// TIA Portal V17 export
// export: Created 2024-09-02T12:50:17.7770543Z, ExportSetting WithDefaults, DisplayName Totally Integrated Automation Portal, DisplayVersion V17, DisplayName TIA Portal Openness, DisplayVersion V17, DisplayName TIA Portal Version Control Interface, DisplayVersion V17, DisplayName STEP 7 Professional, DisplayVersion V17, DisplayName STEP 7 Safety, DisplayVersion V17, DisplayName WinCC Professional, DisplayVersion V17
DATA_BLOCK "SysDI_HMI_SystemInit_OP70"   // DB259
{ DB_Accessible_From_OPC_UA := 'FALSE' }
AUTHOR : OlegFuehrus
FAMILY : HMI
NAME : HMI
VERSION : 0.1
// stored: AutoNumber true, DBAccessibleFromOPCUA false, InstanceOfName SysFB_HMI_SystemInit, InstanceOfType FB
"SysFB_HMI_SystemInit"
   // VAR_INPUT
   //    Start : Bool;
   //    DBNameS7G_Screen1_10 : WString[125];
   //    DBNameS7G_Screen11_20 : WString[125];
   //    DBNameS7G_Screen21_30 : WString[125];
   //    DBNameS7G_Screen31_40 : WString[125];
   //    DBNameS7G_Screen41_50 : WString[125];
   //    DBNameS7G_Screen51_58 : WString[125];
   // END_VAR
   // VAR_IN_OUT
   //    LTLL_Config : "LTLL_typeConfig";
   //    LTLL_Data : "LTLL_typeData";
   //    SYS_StepsHand : "TypeStepsHand";
   //    Finish : Bool;
   // END_VAR
   // VAR RETAIN
   //    s_Counter : Int;
   //    s_SNr : Int;
   //    s_Screen_Nr : Int;
   //    s_Screen_Counter : Int;
   //    s_INIT_ScreenConfig { S7_SetPoint := 'True'} : "LTLL_typeManualConfig";
   //    s_INIT_StepData { S7_SetPoint := 'True'} : "LTLL_typeManualData";
   // END_VAR
BEGIN
END_DATA_BLOCK
